FUNCTION_BLOCK ABSTRACT I_Comm
VAR_INPUT
END_VAR
VAR_OUTPUT
END_VAR
VAR
END_VAR

END_FUNCTION_BLOCK

(* stored: Version 1.1.0.1, ProductVersion 3.1.4024.13
   POU I_Comm: Id {c918bc36-95ef-4710-847f-cd3195d10ef3}, SpecialFunc None *)
